(* cylinder commands *)
TYPE E_CylinderCmd :
(
	Cyl_Idle 		:= 0,// Jog Cylinder command Referance 0 Idle (wait for command)
	Cyl_Init 		:= 1,// Jog Cylinder command Referance 1 initialize Cylinder
	Cyl_Enable 		:= 2,// Jog Cylinder command Referance 2 enable
	Cyl_Disable 	:= 3,// Jog Cylinder command Referance 3 disable
	Cyl_Reset 		:= 4,// Jog Cylinder command Referance 4 reset
	Cyl_Hold 		:= 5,// Jog Cylinder command Referance 5 hold
	Cyl_Teach 		:= 6,// Jog Cylinder command Referance 6 teach timeout settings
	Cyl_Calculate 	:= 7,// Jog Cylinder command Referance 7 calculate timeout settings from parameters
	Cyl_Expand 		:= 8,// Jog Cylinder command Referance 8 expand
	Cyl_Retract 	:= 9 // Jog Cylinder command Referance 9 retract
);
END_TYPE

(* stored: Version 1.1.0.1, ProductVersion 3.1.4022.16
   EnumerationTextList E_CylinderCmd: Id {90e033e9-e3d5-4dc8-8d73-1e41dc41c8fd} *)
